% RSLogix 500 project DIGITALROTAMETER_BAK021.RSS, saved by version 8.30.00.16 %
PROJECT "UNTITLED"    % processor: Bul.1763 MicroLogix 1100 Series B %

PROGRAM FILES
  LAD 2   6 rungs

DATA FILES
  O0 OUTPUT  4 elements
  I1 INPUT  6 elements
  S2 STATUS  66 elements
  B3 BINARY  1 elements
  T4 TIMER  2 elements
  C5 COUNTER  1 elements
  R6 CONTROL  1 elements
  N7 INTEGER  3 elements
  F8 FLOAT  4 elements

LADDER 2
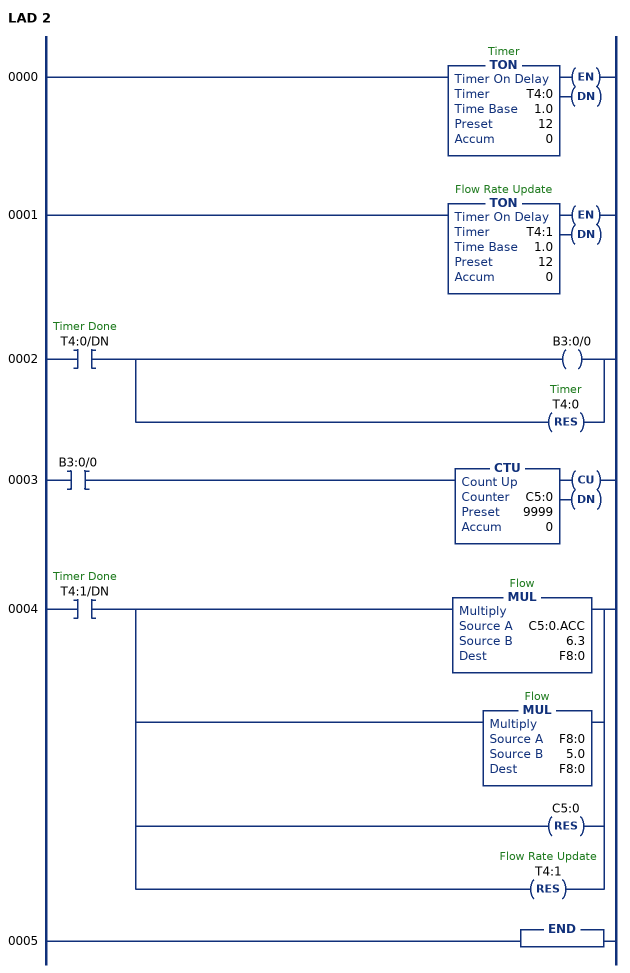
% Rung: 0 %
SOR TON T4:0 1.0 12 0 EOR
%   T4:0  "Timer" %
% Rung: 1 %
SOR TON T4:1 1.0 12 0 EOR
%   T4:1  "Flow Rate Update" %
% Rung: 2 %
SOR XIC T4:0/DN BST OTE B3:0/0 NXB RES T4:0 BND EOR
%   T4:0/DN  "Timer Done" %
%   T4:0  "Timer" %
% Rung: 3 %
SOR XIC B3:0/0 CTU C5:0 9999 0 EOR
% Rung: 4 %
SOR XIC T4:1/DN BST MUL C5:0.ACC 6.3 F8:0 NXB BST MUL F8:0 5.0 F8:0 NXB BST RES C5:0 NXB RES T4:1 BND BND BND EOR
%   T4:1/DN  "Timer Done" %
%   F8:0  "Flow" %
%   T4:1  "Flow Rate Update" %
% Rung: 5 %
SOR END EOR

OTHER DOCUMENTED ADDRESSES
  B3:0/1  "OS"
  B3:0/2  "Timer Reset"
  B3:0/3  "OS"
  B3:0/4  "Update"
  N7:0  "Count"
  N7:1  "Multiply 6.3 Gallons by Count"
  N7:3  "Pulse frequency"

DATA TABLE (non-zero values as saved)
DATA T4
% .PRE .ACC %
% T4:0 % 12 0
% T4:1 % 12 0
DATA C5
% .PRE .ACC %
% C5:0 % 9999 0
